// TIA Portal V17 export
// export: Created 2024-09-02T12:50:37.446963Z, ExportSetting WithDefaults, DisplayName Totally Integrated Automation Portal, DisplayVersion V17, DisplayName TIA Portal Openness, DisplayVersion V17, DisplayName TIA Portal Version Control Interface, DisplayVersion V17, DisplayName STEP 7 Professional, DisplayVersion V17, DisplayName STEP 7 Safety, DisplayVersion V17, DisplayName WinCC Professional, DisplayVersion V17
TYPE "typ_General"
// stored: IsFailsafeCompliant false
   STRUCT
      "Pallet Number" : Int;
      "Variant Number" : Int;
      "HCU ID" : String[25];
      "Pallet Status" : Struct
         "Pallet loaded" : Bool;
         "Global NOK" : Bool;
         Bypass : Bool;
         Repaired : Bool;
         Scraped : Bool;
         Reserve : Bool;
         Reserve_1 : Bool;
         Reserve_2 : Bool;
      END_STRUCT;
      OK_Finished_by : Struct
         OP10 : Bool;
         OP20 : Bool;
         OP30 : Bool;
         OP40 : Bool;
         OP50 : Bool;
         OP60 : Bool;
         OP70_1 : Bool;
         OP70_2 : Bool;
         OP70_3 : Bool;
         Reserve_2 : Bool;
         Reserve_3 : Bool;
         Reserve_4 : Bool;
         Reserve_5 : Bool;
         Reserve_6 : Bool;
         Reserve_7 : Bool;
         Reserve_8 : Bool;
      END_STRUCT;
      Bypass_By : Struct
         OP10 : Bool;
         OP20 : Bool;
         OP30 : Bool;
         OP40 : Bool;
         OP50 : Bool;
         OP60 : Bool;
         OP70_1 : Bool;
         OP70_2 : Bool;
         OP70_3 : Bool;
         Reserve_2 : Bool;
         Reserve_3 : Bool;
         Reserve_4 : Bool;
         Reserve_5 : Bool;
         Reserve_6 : Bool;
         Reserve_7 : Bool;
         Reserve_8 : Bool;
      END_STRUCT;
      Last_Station_Nr : Int;
      NOK_CodeNumber : Int;
      Load_Time : Date_And_Time;
   END_STRUCT;
END_TYPE
